INTERFACE I_TaurusLed

PROPERTY Text : STRING
GET
END_GET
SET
END_SET
END_PROPERTY

END_INTERFACE

(* stored: Version 1.1.0.1, ProductVersion 3.1.4024.12
   Itf I_TaurusLed: Id {849bbff6-f5db-40e4-a15f-bfd252aa8a6a}
   Property Text: Id {63f51548-7e69-4fe1-8400-17ef379a800c}
   Get Get: Id {b5fbbe03-d9c1-45c3-a9db-085bfeddcd17}
   Set Set: Id {8ab33a09-ba33-4097-92d4-3ac64905ff9d} *)
